{attribute 'pack_mode' := '2'}
TYPE ST_FCUFLEX_out :
STRUCT
	CommandForce : INT;
	CommandPosition : WORD;
	PayloadWeight : WORD;
	ControlMode : WORD;
	WeighPayloadNow : WORD;
END_STRUCT
END_TYPE

(* stored: Version 1.1.0.1, ProductVersion 3.1.4024.9
   DUT ST_FCUFLEX_out: Id {308a1ede-6ad9-41c1-8d20-c9f4b720e8fd} *)
